{attribute 'qualified_only'}
VAR_GLOBAL
	Axis1 : Axis_REF;
END_VAR

(* stored: Version 1.1.0.1, ProductVersion 3.1.4024.15
   GVL GVL_Axis: Id {115db183-fd08-4a67-bbee-eeb5f4818801} *)
